RoboDK station: TheWorker.rdk

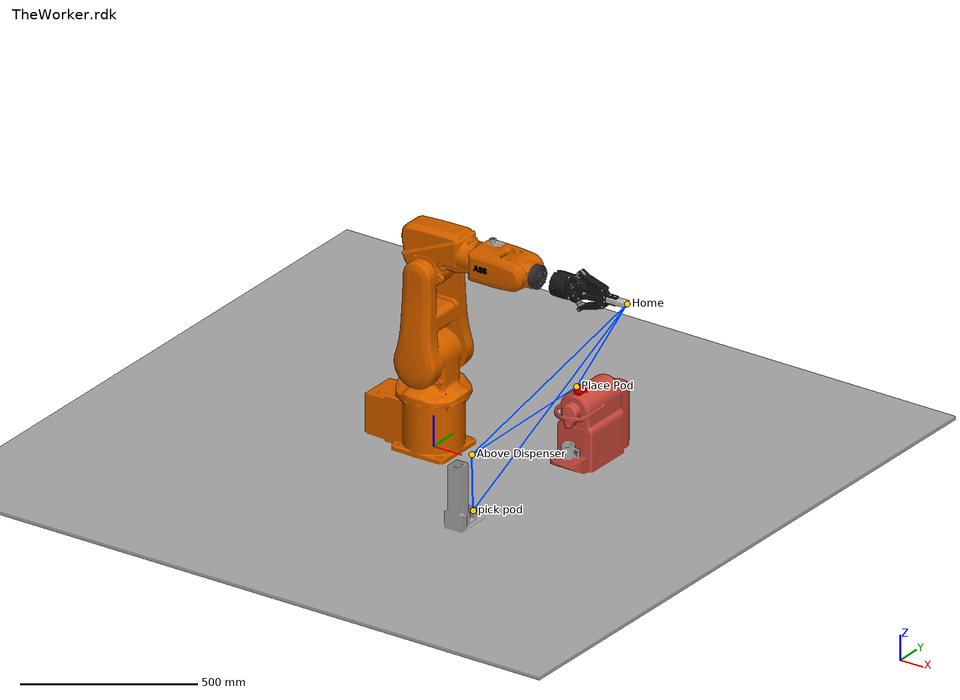
[picture v0: the station drawn from its stored meshes, robots at their saved joint values, targets as dots, program paths as lines]
Station TheWorker (saved by RoboDK 5.6.7). Poses are relative to the parent item; angles as X-Y-Z fixed-axis rotations.
Station parameters (name, value as stored): LIN64
  - frame ABB IRB 120-3/0.6 Base at (-2.05, 0, 0) mm
    - target pick pod (Cartesian target) at (376.12, -343.64, 41.03) mm, rotated rx -179.63 ry -1.29 rz 4.29 deg; joints [-43.236, 48.573, -23.215, 1.337, 64.052, 131.893]
    - target Place Pod (Cartesian target) at (405.24, 123.97, 250.3) mm, rotated rx -178.76 ry 0.51 rz -91.92 deg; joints [16.786, 24.373, -22.849, 0.084, 87.136, 192.491]
    - target Home (Cartesian target) at (664, 0, 630) mm, rotated rx 0 ry 90 rz 0 deg; joints [0, 0, 0, 0, 0, 0]
    - target Above Dispenser (Cartesian target) at (372.26, -344.62, 215.16) mm, rotated rx -179.63 ry -1.29 rz 4.29 deg; joints [-43.653, 58.022, -72.664, 1.244, 104.052, 132.364]
    - robot ABB IRB 120-3/0.6: 6 axes, payload 3 kg, reach 580 mm, repeatability 0.01 mm, weight 25 kg
        modified DH rows (alpha deg, a mm, theta deg, d mm): 0, 0, 0, 290; -90, 0, -90, 0; 0, 270, 0, 0; -90, 70, 0, 302; 90, 0, 0, 0; -90, 0, 180, 72
        joint limits [-165, -110, -90, -160, -120, -400] to [165, 110, 70, 160, 120, 400]; home [0, 0, 0, 0, 0, 0]; saved at [0, 0, 0, 0, 0, 0]
      - tool RobotiQ 2F-140 Gripper (Closed), TCP at (0, 0, 290) mm, size 124 x 75 x 244.3 mm
  - program Flex Test (4 instructions, listed below)
  - program Gripper Test (6 instructions, listed below)
  - object Base Plate at (0, 0, 0) mm, size 2089.3 x 10 x 2040.7 mm, geometry from Base Plate.STL
  - object XN100 at (-170, 200, 0) mm, size 120 x 230 x 317.5 mm, geometry from XN100.STL
  - program attach (9 instructions, listed below)
  - program Prog4 (13 instructions, listed below)
  - object Tazza_VIP_Mauri at (290, -30, 50) mm, size 60.1 x 40.1 x 39.3 mm, geometry from Tazza_VIP_Mauri.stl
  - object Body at (382.29, -291.96, 0) mm, rotated rx 0 ry 0 rz 180 deg, size 68.8 x 120 x 200 mm, geometry from Body.stl
  - object Nsprsocps at (404.76, 148.65, 231.04) mm, rotated rx 158.49 ry 88 rz 62.29 deg, size 29.2 x 37.4 x 37.4 mm, geometry from Nsprsocps.stl
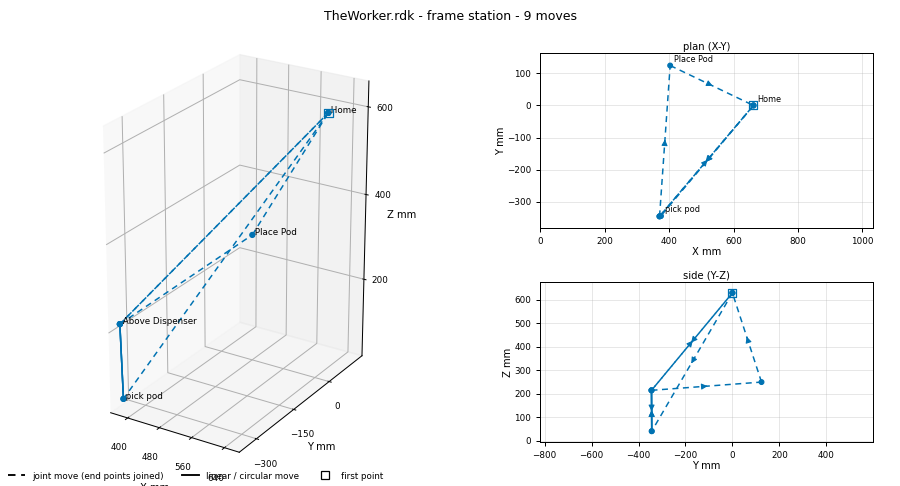
[picture p0: tool path of TheWorker.rdk in frame station, 9 of 19 moves have a stored position in this frame; points joined in program order, loops and branches not executed]

--- program Flex Test ---
  Set Ref.: Frame 3 at (-455.88, 959.54, 600.03) mm, rotated rx 88.8 ry 4.28 rz -4.88 deg
  MoveJ (Home) [its target is no longer in the station]
  MoveJ (Flex) [its target is no longer in the station]
  MoveJ (Home) [its target is no longer in the station]

--- program Gripper Test ---
  Set Ref.: Frame 3 at (-455.88, 959.54, 600.03) mm, rotated rx 88.8 ry 4.28 rz -4.88 deg
  Set Tool: RobotiQ 2F-140 Gripper (Closed) at (0, 0, 290) mm
  MoveJ (Home) [its target is no longer in the station]
  Run GripperTesting
  Pause 20.0 s
  MoveJ (Flex) [its target is no longer in the station]

--- program attach ---
  Set Ref.: Frame 3 at (-355.88, 959.54, 600.02) mm, rotated rx 88.8 ry 4.28 rz -4.88 deg
  Set Tool: RobotiQ 2F-140 Gripper (Closed) at (0, 0, 290) mm
  MoveJ (Home) [its target is no longer in the station]
  MoveJ (Target 7) [its target is no longer in the station]
  Attach to RobotiQ 2F-140 Gripper (Closed)
  MoveJ (Home) [its target is no longer in the station]
  MoveJ (Target 6) [its target is no longer in the station]
  Detach from RobotiQ 2F-140 Gripper (Closed)
  MoveJ (Home) [its target is no longer in the station]

--- program Prog4 ---
  Set Ref.: ABB IRB 120-3/0.6 Base
  Set Tool: RobotiQ 2F-140 Gripper (Closed) at (0, 0, 290) mm
  MoveJ (Home)
  MoveJ (pick pod)
  Attach to RobotiQ 2F-140 Gripper (Closed)
  MoveL (Above Dispenser)
  MoveJ (Place Pod)
  MoveJ (Home)
  MoveJ (Above Dispenser)
  MoveL (pick pod)
  Detach from RobotiQ 2F-140 Gripper (Closed)
  MoveL (Above Dispenser)
  MoveJ (Home)
